FUNCTION_BLOCK GreenMasterDO_Base
VAR_IN_OUT
	DOut: DigitalOutputs;
END_VAR
VAR_INPUT
	H_GP1: BOOL;
	C_GP1: BOOL;
	ExhaustRunning: BOOL;
	F_QM1: BOOL;
	T_QM3: BOOL;
	R_QM1: BOOL;
	F_QM2: BOOL;
	SupplyRunning: BOOL;
	T_QM1_1: BOOL;
	T_QM1_2: BOOL;
	T_QM1_3: BOOL;
	T_QM1_4: BOOL;
	T_QM1_5: BOOL;
	T_QM1_6: BOOL;			
	AlarmRelayA: BOOL;
	AlarmRelayB: BOOL;
	AlarmRelayC: BOOL;
	AlarmRelayD: BOOL;
END_VAR
VAR_OUTPUT
END_VAR
VAR
END_VAR

END_FUNCTION_BLOCK

(* stored: Version 1.1.0.1, ProductVersion 3.1.4024.4
   POU GreenMasterDO_Base: Id {5ad275aa-23a9-47d4-b009-c6105067168f}, SpecialFunc None *)
